(* PLC project fbs-datalayer-subscriptions-settings.project, Rexroth ctrlX PLC Engineering ctrlX PLC 2.1.0 *)
(* stored: creationDateTime 2023-07-13T10:31:13.7872699, modificationDateTime 2023-07-13T10:29:01.8718689 *)

PROGRAM PLC_PRG
  VAR
    bStart_read : BOOL := TRUE;
    bStart_write : BOOL;
    bExecute_read : BOOL;  (* Read values *)
    fbDL_ReadNodeValue : DL_ReadNodeValue;
    bActive_read : BOOL;
    bDone_read : BOOL;
    DataRead : DL_NodeValue;
    bErrorRead : BOOL;
    ErrorIDRead : ERROR_CODE;
    ErrorIdent_read : ERROR_STRUCT;
    fbR_TRIG_read : R_TRIG;
    fbFlatbuffer : comm_datalayer_SubscriptionSettings;
    iRead_X : INT;
    iRead_Y : INT;
    iRead_Z : INT;
    iRead : INT;
    fbBuilder : FlatBufferBuilder;  (* Write values *)
    maximumBufferSize : UDINT;
    iWritten : INT;
    bExecute_write : BOOL;
    fbDL_WriteNodeValue : DL_WriteNodeValue;
    bActive_write : BOOL;
    bDone_write : BOOL;
    fbValueIn : DL_NodeValue;
    fbValueOut : DL_NodeValue;
    bError_write : BOOL;
    ErrorID_write : ERROR_CODE;
    ErrorIdent_write : ERROR_STRUCT;
    fbR_TRIG_write : R_TRIG;
    strNodePath : STRING(255) := 'datalayer/subscriptions/settings';
  END_VAR

                  IF bStart_read THEN
	bStart_read := FALSE;
	bExecute_read := TRUE;	
END_IF


fbDL_ReadNodeValue(
	Execute:= bExecute_read,
	Done=> bDone_read,
	Active=> bActive_read,
	Error=> bErrorRead,
	ErrorID=> ErrorIDRead,
	ErrorIdent=> ErrorIdent_read,
	ClientId:= ,
	NodeName:= strNodePath,
	NodeValue:= DataRead);

IF bDone_read AND bExecute_read THEN
	bExecute_read := FALSE;

	fbFlatbuffer.getRootAsSubscriptionSettings(data:=
	DataRead.GetData(), size:= DataRead.GetSize());
	
	maximumBufferSize := fbFlatbuffer.getMaximumBufferSize();
		
	bStart_write := TRUE;
END_IF

	
IF bStart_write THEN
	bStart_write := FALSE;

	maximumBufferSize := (maximumBufferSize + 1);
	IF maximumBufferSize > 55 THEN
		maximumBufferSize := 50;
	END_IF
	
	fbBuilder(forceDefaults := TRUE);
	fbFlatbuffer.startSubscriptionSettings(fbBuilder);
	
	fbFlatbuffer.addMaximumBufferSize(maximumBufferSize);
	
	fbBuilder.finish(fbFlatbuffer.endSubscriptionSettings());
	fbValueIn.SetFlatbuffer(fbBuilder);
	
	bExecute_write := TRUE;
END_IF

	
fbDL_WriteNodeValue(
	Execute:= bExecute_write,
	Done=> bDone_write,
	Active=> bActive_write,
	Error=> bError_write,
	ErrorID=> ErrorID_write,
	ErrorIdent=> ErrorIdent_write,
	ClientId:= ,
	NodeName:= strNodePath,
	NodeValueIn:= fbValueIn,
	NodeValueOut:= fbValueOut);

IF bDone_write AND bExecute_write THEN
	bExecute_write := FALSE;	
	iWritten := iWritten + 1;
	
	bStart_read := TRUE;
END_IF
	

                
END_PROGRAM

CONFIGURATION Application
  RESOURCE Application ON PLC
    TASK MainTask(INTERVAL := T#2000ms, PRIORITY := 30);
    PROGRAM PLC_PRG WITH MainTask : PLC_PRG;
  END_RESOURCE
END_CONFIGURATION
